FUNCTION F_RangeSetpoint : BOOL
VAR_INPUT
	lrSetpoint: LREAL;
	lrActValue: LREAL;
	lrRangePercent: LREAL;
END_VAR
VAR
	lrTempSetpointUp: LREAL;
	lrTempSetpointDown: LREAL;
END_VAR

F_RangeSetpoint:=FALSE;

lrTempSetpointDown:=lrSetpoint-(lrSetpoint*(lrRangePercent/100.0));
lrTempSetpointUp:=lrSetpoint+(lrSetpoint*(lrRangePercent/100.0));

IF (lrActValue>=lrTempSetpointDown) AND (lrActValue<=lrTempSetpointUp) THEN
	F_RangeSetpoint:=TRUE;
END_IF

END_FUNCTION

(* stored: Version 1.1.0.1, ProductVersion 3.1.4024.4
   POU F_RangeSetpoint: Id {f6c276bf-ceeb-4732-9949-a441b5b5ac1f}, SpecialFunc None *)
